FUNCTION_BLOCK CM_DO_CALL
VAR_INPUT
END_VAR
VAR_OUTPUT
END_VAR
VAR
END_VAR

// NETWORK 1

END_FUNCTION_BLOCK

(* stored: Version 1.1.0.1, ProductVersion 3.1.4024.13
   POU CM_DO_CALL: Id {53aa745f-c1c2-4143-b381-f436608fe08c}, SpecialFunc None *)
